{attribute addProperty BoxType "KL8610"}
{attribute addProperty Id "KL8601_1KL_B0A8062F00"}
{attribute addProperty CRC "151672865"}
{attribute addProperty SizeInBites "0"}
{attribute addProperty SizeInBytes "0"}
TYPE KL8610_090A5821 :
STRUCT
	{attribute addProperty Name "KL8601_1"}
	KL8601_1 : KL_B0A8062F;
END_STRUCT
END_TYPE

(* stored: Version 1.2.0.0, ProductVersion 3.1.4024.9
   DUT KL8610_090A5821: Id {57933a84-e08a-489a-b2ed-7686c32bff28} *)
